FUNCTION_BLOCK FB_ShippingRobot_PhotoStandByPos EXTENDS FB_RobotRegionMove_BufferArea
VAR_INPUT
	Input	: REFERENCE TO ST_InputTable;
	Output	: REFERENCE TO ST_OutputTable;
END_VAR
VAR_OUTPUT
END_VAR
VAR
	// 用於轉型 Lreal
	iCmdPosA	: INT;
	
	TON_RobotActionTimeOut		: TON;
	TON_CheckRobotDoneTimeOut	: TON;
	
END_VAR

THIS^.A00_BasicUnits();
SUPER^.A10_StateControl();

Area := E_RobotArea.ShippingCCDPos;

ACTION A00_BasicUnits:
TON_RobotActionTimeOut( PT := T#60S);
TON_CheckRobotDoneTimeOut(PT := T#30S);
END_ACTION

METHOD M_CheckCommandVaild : BOOL
VAR_INPUT
END_VAR
VAR
END_VAR
THIS^.Get :=Info.Get;
UseA := Info.UseA;
UseB := Info.UseB;

// 出貨區小手臂只有 A爪,所以程式內只有判斷 useA
IF UseB THEN
	M_CheckCommandVaild := FALSE;
	status 				:= 'FB_ShippingRobot_PhotoStandByPos: WrongCommand not have B Clamp , not can retry';
	RETURN;
END_IF
IF NOT UseA THEN
	M_CheckCommandVaild := FALSE;
	status 				:= 'FB_ShippingRobot_PhotoStandByPos: WrongCommand A Clamp must be used';
	RETURN;
END_IF

//
IF info.A_Position <> 0 THEN
	M_CheckCommandVaild := TRUE;
	status				:= 'FB_ShippingRobot_PhotoStandByPos: WrongCommand not have Position';
END_IF

M_CheckCommandVaild := TRUE;
END_METHOD

METHOD  M_STATE_ABORTED
VAR_INPUT
END_VAR

Busy  := FALSE;
Error := TRUE;
Aborted := TRUE;
uiAbortingStep 	:= 0;
_AbortCompleted := FALSE;

// 狀態機切換
IF NOT Execute THEN
	eState := STATE_RESETTING;
ELSIF Execute AND reset THEN
	Error	:= false;
	Aborted	:= false;
	eState 	:= STATE_EXECUTING;
END_IF
END_METHOD

METHOD  M_STATE_ABORTING
VAR_INPUT
END_VAR

CASE uiAbortingStep OF
	0 :
		_Abort := FALSE;
		TON_RobotActionTimeOut.IN 	 := FALSE;
		TON_CheckRobotDoneTimeOut.IN := FALSE;
		
		uiAbortingStep:=9999;

	9999:	
		_AbortCompleted:=TRUE;
END_CASE

IF _AbortCompleted THEN	
	eSTATE :=STATE_ABORTED;
END_IF
END_METHOD

METHOD  M_STATE_DONE
VAR_INPUT
END_VAR

Busy := FALSE;
Done := TRUE;
IF NOT Execute THEN
    eState := STATE_RESETTING;
END_IF
END_METHOD

METHOD  M_STATE_DORMANT
VAR_INPUT
END_VAR
Busy 			:= FALSE;
Done 			:= FALSE;
Aborted 		:= FALSE;
Error			:= FALSE;
Paused			:= FALSE;
ErrorID			:= 0;
Status			:= '';
UniqueErrorCode := '';

_Executed 			:= FALSE;
_Error				:= FALSE;
_Abort				:= FALSE;
_ResetCompleted 	:= FALSE;
_AbortCompleted 	:= FALSE;
_HoldingCompleted 	:= FALSE;
_HeldCompleted	 	:= FALSE;
_UnholdCompleted 	:= FALSE;

uiExecutingStep 		:= 0;
uiResettingStep 		:= 0;
uiAbortingStep 			:= 0;
uiHoldingStep			:= 0;
uiHeldStep				:= 0;
uiUnholdStep			:= 0;

TON_RobotActionTimeOut.IN 	 := FALSE;
TON_CheckRobotDoneTimeOut.IN := FALSE;

IF Execute THEN
    eState := STATE_EXECUTING;
END_IF
END_METHOD

METHOD  M_STATE_ERROR
VAR_INPUT
END_VAR

ERROR   := TRUE;
Busy	:= FALSE;
_Error	:= false;

IF NOT Execute THEN	
	Error	:= FALSE;
	eSTATE	:=STATE_RESETTING;
END_IF
END_METHOD

METHOD  M_STATE_EXECUTING
VAR_INPUT
END_VAR
VAR_INST
	Address_A	 : INT;
	BoxReady_1st : BOOL;
END_VAR
busy := true;

// 暫停
IF Pause THEN 
	_HoldingCompleted 	:= FALSE;
	_HeldCompleted	 	:= FALSE;
	_UnholdCompleted 	:= FALSE;
	uiHoldingStep		:= 0;
	uiHeldStep			:= 0;
	uiUnholdStep		:= 0;
	eState    			:= STATE_Holding;
END_IF

// 動作主流程 狀態機
CASE uiExecutingStep OF
	
	0:		// 檢查命令是否是有效值
			IF M_CheckCommandVaild() THEN
				uiExecutingStep := 1000;
			ELSE
				_Error := TRUE;
			END_IF
			
	1000:	
			uiExecutingStep := 10000;
			
	10000:	// RobotAction
			TON_RobotActionTimeOut.IN := TRUE;
			IF NOT Robot._DI1.Done THEN  
			
					 Robot.M_StartRobotAbsMove(GetBox:=TRUE,
												UseClampA:=UseA,
												UseClampB:=FALSE,
												Area:=Area,
												ClampA_Address:=0,
												ClampB_Address:=0,
												BoxReady_1:=BoxReady_1st,
												BoxReady_2:=FALSE);	  
				
			ELSE
				uiExecutingStep := 11000;
			END_IF
			
			IF TON_RobotActionTimeOut.Q THEN
				_Abort 	:= TRUE;
				Status	:= 'FB_ShippingRobot_PhotoStandByPos Step 10000: RobotAction Timeout,can retry';
			END_IF
			
	11000:	// reset 手臂命令
			Robot.M_ResetRobotAbsMove(UseA,UseB); // Clear command and go to place box
			TON_RobotActionTimeOut.IN 	 := FALSE;
			TON_CheckRobotDoneTimeOut.IN := TRUE;
			IF NOT Robot._DI1.Done THEN
				TON_CheckRobotDoneTimeOut.IN := FALSE;
            	uiExecutingStep := 90000; 
        	END_IF
			IF TON_CheckRobotDoneTimeOut.Q THEN
				_Error := TRUE;
				status := 'FB_ShippingRobot_PhotoStandByPos Step 11000: Wait Robot done Timeout';
			END_IF
		
	90000:
			Status    := 'FB_ShippingRobot_PhotoStandByPos Step 90000: Process completed';
        	_Executed := TRUE;
end_case

// 狀態機切換
IF NOT Execute THEN
	eState := STATE_RESETTING;
ELSIF _Error THEN
	eState := STATE_ERROR;
ELSIF _Abort THEN
	eState := STATE_ABORTING;
ELSIF _Executed THEN
	eState := STATE_DONE;
END_IF
END_METHOD

METHOD M_STATE_HELD
VAR_INPUT
END_VAR

Busy 	:= FALSE;
Paused 	:= TRUE;

CASE uiHeldStep OF
	0:
		uiHeldStep := 9999;

	9999:
		_HeldCompleted := TRUE;	

END_CASE

IF _HeldCompleted AND NOT Pause THEN
	eState := STATE_UnHold;
END_IF
END_METHOD

METHOD M_STATE_HOLDING
VAR_INPUT
END_VAR

CASE uiHoldingStep OF 
	0:	// 需關閉 Timer 等等須暫停的變數
		TON_RobotActionTimeOut.IN 	 := FALSE;
		TON_CheckRobotDoneTimeOut.IN := FALSE;
		
		uiHoldingStep := 9999;
		
	9999:	// holding 完成
		_HoldingCompleted := TRUE;
END_CASE

IF _HoldingCompleted THEN
	eState := STATE_Held;
END_IF
END_METHOD

METHOD  M_STATE_RESETTING
VAR_INPUT
END_VAR

Busy := TRUE;
Error := FALSE;
_Error := FALSE;

CASE uiResettingStep OF

	0:
		uiResettingStep := 9999;

	9999:
		Done := FALSE;
		Busy := FALSE;
		_ResetCompleted:=TRUE;
END_CASE

IF _ResetCompleted THEN
	eSTATE:=STATE_DORMANT;
END_IF
END_METHOD

METHOD M_STATE_UNHOLD
VAR_INPUT
END_VAR
CASE uiUnholdStep OF 
	0:		
		uiUnholdStep := 9999;
		
	9999:
		_UnholdCompleted := TRUE;
		
END_CASE

IF _UnholdCompleted THEN
	Paused := FALSE;
	eState := STATE_EXECUTING;
END_IF
END_METHOD

END_FUNCTION_BLOCK

(* stored: Version 1.1.0.1, ProductVersion 3.1.4024.13
   POU FB_ShippingRobot_PhotoStandByPos: Id {a3d3a693-3945-4127-aa26-6a5787fd5c1b}, SpecialFunc None
   Folder Method: Id {cfe556f2-c6f1-4541-8468-72036bf50279}
   Folder STATE: Id {5a6dde8e-dce0-4b4d-8e95-dfd42796c57d}
   Action A00_BasicUnits: Id {f575c56b-7b11-4743-aff0-1fc3bdb25e89}
   Method M_CheckCommandVaild: Id {d55f611e-7059-488c-9ef8-136d00f45de9}
   Method M_STATE_ABORTED: Id {2ae87bb4-5196-4a4c-9c74-79fd18991d47}
   Method M_STATE_ABORTING: Id {b280392d-c6a5-4020-9def-104084606ecd}
   Method M_STATE_DONE: Id {c07569e4-f388-4922-af7c-41d2ca428863}
   Method M_STATE_DORMANT: Id {16f1c610-6700-4f0b-96ec-1d452d4bad2b}
   Method M_STATE_ERROR: Id {adb52bf2-bd12-481c-913c-20a498bcca32}
   Method M_STATE_EXECUTING: Id {c82398c3-4a0b-4a02-92ad-4e93f82c71d3}
   Method M_STATE_HELD: Id {98572061-20a5-4ed4-98b2-759d1197576a}
   Method M_STATE_HOLDING: Id {eb9e8942-dca8-447d-a17d-2b16895eb943}
   Method M_STATE_RESETTING: Id {a149e4c4-8485-4bca-b06a-12c330366d7d}
   Method M_STATE_UNHOLD: Id {7b89ee00-48ee-416a-b6db-b8e5e24a2ef8} *)
